	roboArmStates.stUInsertBackStart:		
		uInsertBack  := TRUE;
		resetActive  := TRUE;
		nextState(roboArmStates.stUInsertBackMove);				
		
// *** Unload Insert Back - Move
// Задава се програма на робота

	roboArmStates.stUInsertBackMove:		
		Stations.roboData := dataRequestRobot.roboPrg_PreUnload;		
		nextState(roboArmStates.stUInsertBackMoveCheck);		
		
// *** Unload Insert Back - Move Check
// Робота изпълни ли си хода ?

	roboArmStates.stUInsertBackMoveCheck:
		IF Stations.roboData = dataRequestRobot.done THEN				
		    nextState(roboArmStates.stUInsertBackSync);		
		END_IF		
		IF Stations.roboData = dataRequestRobot.error THEN
			nextState(roboArmStates.stErrRobot);
		END_IF
		timeOutError(robotMoveTime, roboArmStates.stErrRobotTimeOut);

// *** Unload Insert Back - Sync

	roboArmStates.stUInsertBackSync:	
		depWait(globalDeps.depULoadRobotOutOfRich);	     			
		nextState(roboArmStates.stUInsertBackDone);				
		
// *** Unload Insert Back - Done

	roboArmStates.stUInsertBackDone:
        uInsertBack	:= FALSE;
		nextState(roboArmStates.stUnloadStart);		
	
// *** Step Mode
		
	roboArmStates.stStepBlock:
		setDisplayState(roboArmDisplayStates.dStWaitForNextStep);
		
// *** Stop 
// Станията е деактивирана
	
	roboArmStates.stStop:
	
		initDone			  := FALSE; 			
		resetActive           := FALSE;                           
		nextMoveStart         := FALSE;                            
		moveToEmptyStart      := FALSE;                           
		emptyToUnloadStart    := FALSE;                           
		unloadPalletStart     := FALSE;                            
		loadPalletStart       := FALSE;                            
		emptyPosStart         := FALSE;                            
		loadStart             := FALSE;                            
		unloadStart           := FALSE;                            
		lInsertStart          := FALSE;                            
		lInsertLockStart      := FALSE;                 
		lInsertBack           := FALSE;             
		uInsertStart          := FALSE;                           
		uInsertLockStart      := FALSE;                          
		uInsertBack           := FALSE;         
		blockRunForLoad       := FALSE;
		
// *** ERRORS

// *** ERROR - Init Sensor
// При стартиране на програмата не трябва да има сензор в грипера на робота
		roboArmStates.stErrInitSensor:
			setDisplayState(roboArmDisplayStates.dStErrInitSensorInGrip);
			
// *** ERROR - Pallet On 24
// При стартиране на програмата не трябва да има тара на чакаща поз. HEX 24
		roboArmStates.stErrInitPalletOn24:
			setDisplayState(roboArmDisplayStates.dStErrInitPalletOnWaitPos24);			

// *** ERROR - Pallet On 27
// При стартиране на програмата не трябва да има тара на чакаща поз. HEX 27
		roboArmStates.stErrInitPalletOn27:
			setDisplayState(roboArmDisplayStates.dStErrInitPalletOnWaitPos27);		

// *** ERROR - Grip Not Open
// Гирипера на робота не е отворил навреме
		roboArmStates.stErrGripNotOpen:
			setDisplayState(roboArmDisplayStates.dStErrGripNotOpen);
	
// *** ERROR - Grip Not Close
// Гирипера на робота не е затворил навреме
		roboArmStates.stErrGripNotClose:
			setDisplayState(roboArmDisplayStates.dStErrGripNotClose);			
			
// *** ERROR - Rot Not turn 180
// Ротатора не е завъртял сензора на обратно (180 град.)
		roboArmStates.stErrRotNotTurn180:
			setDisplayState(roboArmDisplayStates.dStErrRotatorNotTurn180);			
			
// *** ERROR - Rot Not turn 0
// Ротатора не е завъртял сензора (0 град.)
		roboArmStates.stErrRotNotTurn0:
			setDisplayState(roboArmDisplayStates.dStErrRotatorNotTurn0);					
			
// *** ERROR - Slinde Not Down
// Слайдера който захваща тарата не в долна поз.
		roboArmStates.stErrSlliderNotDown:
			setDisplayState(roboArmDisplayStates.dStErrSlideNotDown);			
			
// *** ERROR - Slinde Not Up
// Слайдера който захваща тарата не в горна поз.
		roboArmStates.stErrSlideNotUp:
			setDisplayState(roboArmDisplayStates.dStErrSlideNotUp);	

// *** ERROR - Robot Error
// Има някаква грашка върната от робот контролера
		roboArmStates.stErrRobot:	
			setDisplayState(roboArmDisplayStates.dStErrRobotError);	
		
// *** ERROR - Robot Reset
// Времето за изпълнение на HOME програмата на работа е отнело трвърде мн.
		roboArmStates.stErrRobotReset:	
			setDisplayState(roboArmDisplayStates.dStErrRobotHomeMoveIsTooLong);			

// *** ERROR - Robot Time out
// Времето за изпълнение на движение на робота е отнело твърде мн.
		roboArmStates.stErrRobotTimeOut:	
			setDisplayState(roboArmDisplayStates.dStErrRobotMoveIsTooLong);	

// *** ERROR - Robot Recipe TimeOut
// Времето за зареждане на рецепта в робота е отнело твърде мн.
		roboArmStates.stErrRobotRecipeTimeOut:	
			setDisplayState(roboArmDisplayStates.dStErrRobotRecipeLoadIsTooLong);		
		
// *** ERROR - Robot Wait Pos Pallet Fail
// На мястото на чакащата поз. няма тара
		roboArmStates.stErrNoPalletWaitPos:	
			setDisplayState(roboArmDisplayStates.dStErrRobotWaitPosIsEmpty);	

// *** ERROR - Paallet On Wait Pos
// Робота трябва да занесе тара на чакаща поз, но там вече има
		roboArmStates.stErrPalletOnWaitPos:			
			setDisplayState(roboArmDisplayStates.dStErrRobotWaitPosIsNotEmpty);			
			
// *** ERROR - No Pallet Unload
// Робота не е могъл да вдигне или е изпуснал тара
		roboArmStates.stErrNoPalletUnload:	
			setDisplayState(roboArmDisplayStates.dStErrRobotNoPalletAtUnloadStacker);
			unloadPalletStart := FALSE;
			palletIn          := FALSE;	
			
// *** EMG State					
	roboArmStates.stEMG: 
		nextState(roboArmStates.stInit);

END_CASE

METHOD PRIVATE signalLamps
VAR_INPUT
	
	enable      : BOOL;                  
	lamp24      : BOOL;                  // Активиране на лампа за чакаща поз. за HEX 24
	sensor24    : BOOL;                  // Сигнал от сензора за поставена тара на поз. HEX 24
	lamp27      : BOOL;                  // Активиране на лампа за чакаща поз. за HEX 24	
	sensor27    : BOOL;                  // Сигнал от сензора за поставена тара на поз. HEX 27

END_VAR

VAR
	
	lamp24On    : BOOL;
	lamp27On    : BOOL;
	
END_VAR
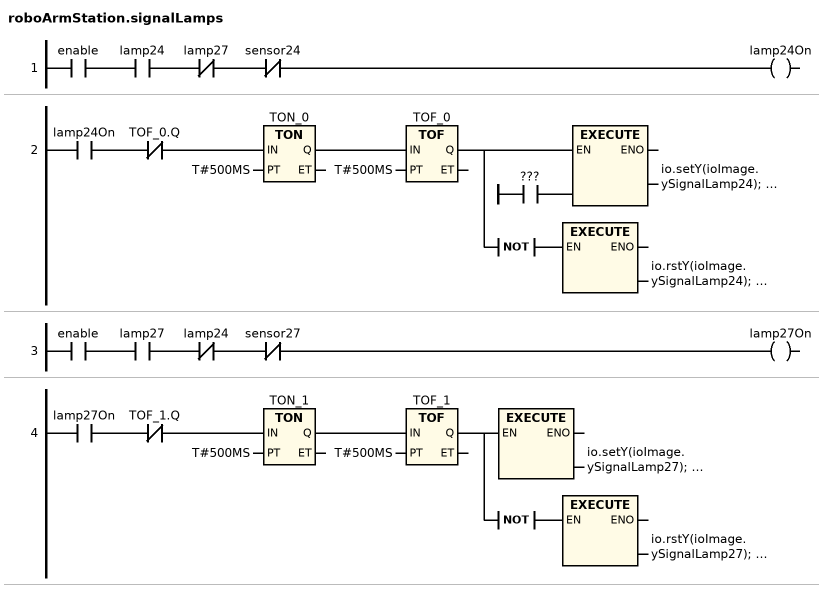
// NETWORK 1
lamp24On := enable AND lamp24 AND NOT lamp27 AND NOT sensor24;

// NETWORK 2
TON_0(IN := lamp24On AND NOT TOF_0.Q, PT := T#500MS); // TON
TOF_0(IN := TON_0.Q, PT := T#500MS); // TOF
IF TOF_0.Q THEN io.setY(ioImage.ySignalLamp24); END_IF
IF NOT TOF_0.Q THEN io.rstY(ioImage.ySignalLamp24); END_IF

// NETWORK 3
lamp27On := enable AND lamp27 AND NOT lamp24 AND NOT sensor27;

// NETWORK 4
TON_1(IN := lamp27On AND NOT TOF_1.Q, PT := T#500MS); // TON
TOF_1(IN := TON_1.Q, PT := T#500MS); // TOF
IF TOF_1.Q THEN io.setY(ioImage.ySignalLamp27); END_IF
IF NOT TOF_1.Q THEN io.rstY(ioImage.ySignalLamp27); END_IF
END_METHOD

END_FUNCTION_BLOCK

// ---- POUs/ROBOT.TcPOU
PROGRAM Robot
VAR
	fbRobot						: FB_Robot_Mitsubishi;
	nCurrentState				: DINT;
	nLastState					: DINT;				
	rtRobot_ProgramStarted		: TON;
	rtRobot_ProgramCompleted	: TON;
	fbTimerRobot				: TON;
	gbTimerTimeoutRobot			: TON;
END_VAR

Stations.gstRobotMitsubishi.sRobotAddress := '192.168.0.20';
Stations.gstRobotMitsubishi.nRobotPort := 10004;
Stations.gstRobotMitsubishi.bAutomaticMode := TRUE;
fbRobot(Robot := Stations.gstRobotMitsubishi,
	PacketManager := Stations.gstRobotMitsubishiPacketManager);
		
rtRobot_ProgramStarted(IN:=NOT Stations.gstRobotMitsubishi.bReady 
						AND NOT Stations.gstRobotMitsubishi.bProgramCompleted, PT:=T#30MS);
rtRobot_ProgramCompleted(IN:= Stations.gstRobotMitsubishi.bReady AND Stations.gstRobotMitsubishi.bProgramCompleted 
							AND Stations.gstRobotMitsubishi.nDependencyState = 0, PT:=T#30MS);

// If robot error
IF Stations.gstRobotMitsubishi.bError 
AND nCurrentState > E_RobotStates.STATE_INIT_CHECK_ROBOT_ERROR_DONE 
AND nCurrentState < E_RobotStates.STATE_ERROR THEN
	nLastState:=nCurrentState;
	nCurrentState:=E_RobotStates.STATE_ERROR;
END_IF
//Statuses
TagsRobot.robotError := Stations.gstRobotMitsubishi.bError;
TagsRobot.robotComOnline := Stations.gstRobotMitsubishi.bOnline;

// Robot Settings
Stations.gstRobotMitsubishi.nTargetProductID := TagsRobot.roboRecipeNum;
Stations.gstRobotMitsubishi.nTargetGripperID := 1;		//TBD Setting for GipperID
Stations.gstRobotMitsubishi.nTargetTrayOrientation := TagsRobot.rotPallet;
		
CASE nCurrentState OF
	E_RobotStates.STATE_WAITING_FOR_INIT:
		IF Stations.roboData = dataRequestRobot.roboInit THEN			
			nLastState := nCurrentState;
			nCurrentState := E_RobotStates.STATE_INIT_ROBOT_TOGGLE;
		END_IF
		
	E_RobotStates.STATE_INIT_ROBOT_TOGGLE:
		IF Stations.gstRobotMitsubishi.bAutomaticMode THEN
			Stations.gstRobotMitsubishi.bDoReset:=FALSE;
			Stations.gstRobotMitsubishi.bToggleConnect:=FALSE;
			Stations.gstRobotMitsubishi.bDoStart:=FALSE;
			fbTimerRobot(IN:=TRUE,PT:=T#1000MS);
			IF fbTimerRobot.Q THEN
				fbTimerRobot(IN:=FALSE);				
				nLastState := nCurrentState;
				nCurrentState :=E_RobotStates.STATE_INIT_ROBOT_ON;
			END_IF
		ELSE
			// Robot Auto  = true
		END_IF

	E_RobotStates.STATE_INIT_ROBOT_ON:
		IF Stations.gstRobotMitsubishi.bOnline THEN
			nLastState := nCurrentState;
			nCurrentState :=E_RobotStates.STATE_INIT_CHECK_ROBOT_ERROR;
		ELSE
			Stations.gstRobotMitsubishi.bToggleConnect:=TRUE;
			a_ToggleRobot();
		END_IF	

	E_RobotStates.STATE_INIT_CHECK_ROBOT_ERROR:
		IF Stations.gstRobotMitsubishi.bError OR Stations.gstRobotMitsubishi.nCurrentState = E_Robot_Mitsubishi_States.STATE_WAITING_RESET THEN
			Stations.gstRobotMitsubishi.bDoReset:=TRUE;
			nLastState := nCurrentState;
			nCurrentState :=E_RobotStates.STATE_INIT_CHECK_ROBOT_ERROR_DONE;
		ELSE
			nLastState := nCurrentState;
			nCurrentState :=E_RobotStates.STATE_INIT_CHECK_ROBOT_READY;
		END_IF	
	
	E_RobotStates.STATE_INIT_CHECK_ROBOT_ERROR_DONE:
		IF Stations.gstRobotMitsubishi.nCurrentState = E_Robot_Mitsubishi_States.STATE_OPERATIONAL THEN
			IF NOT Stations.gstRobotMitsubishi.bError THEN
				nLastState := nCurrentState;
				nCurrentState :=E_RobotStates.STATE_INIT_CHECK_ROBOT_READY;
			ELSE
				a_ToggleRobot();
			END_IF
		ELSIF Stations.gstRobotMitsubishi.nCurrentState = E_Robot_Mitsubishi_States.STATE_WAITING_RESET THEN
			nLastState := nCurrentState;
			nCurrentState :=E_RobotStates.STATE_INIT_CHECK_ROBOT_ERROR;
		END_IF
		
	E_RobotStates.STATE_INIT_CHECK_ROBOT_READY:
		IF NOT Stations.gstRobotMitsubishi.bReady OR NOT Stations.gstRobotMitsubishi.bExecuting THEN
			Stations.gstRobotMitsubishi.bDoStart:=TRUE;
			nLastState := nCurrentState;
			nCurrentState :=E_RobotStates.STATE_INIT_CHECK_ROBOT_READY_DONE;		
		ELSE
			nLastState := nCurrentState;
			nCurrentState :=E_RobotStates.STATE_INIT_CHECK_ROBOT_SERVOON;	
		END_IF
	
	E_RobotStates.STATE_INIT_CHECK_ROBOT_READY_DONE:
		IF Stations.gstRobotMitsubishi.bReady AND Stations.gstRobotMitsubishi.bExecuting THEN
			nLastState := nCurrentState;
			nCurrentState :=E_RobotStates.STATE_INIT_CHECK_ROBOT_SERVOON;
		ELSE
			a_ToggleRobot();					
		END_IF
				
	E_RobotStates.STATE_INIT_CHECK_ROBOT_SERVOON:		
		IF Stations.gstRobotMitsubishi.bPoweredOn AND Stations.gstRobotMitsubishi.bReady THEN
			nLastState := nCurrentState;
			nCurrentState :=E_RobotStates.STATE_INIT_DONE;
		ELSE 				
			Stations.gstRobotMitsubishi.bDoServoOn:=TRUE;
			nLastState := nCurrentState;
			nCurrentState :=E_RobotStates.STATE_INIT_CHECK_ROBOT_SERVOON_DONE;
		END_IF
		
	E_RobotStates.STATE_INIT_CHECK_ROBOT_SERVOON_DONE:
		IF Stations.gstRobotMitsubishi.bPoweredOn AND Stations.gstRobotMitsubishi.bReady THEN
			nLastState := nCurrentState;
			nCurrentState :=E_RobotStates.STATE_INIT_DONE;
		END_IF	
		
	E_RobotStates.STATE_INIT_DONE:
		Stations.roboData := dataRequestRobot.done;
		nLastState := nCurrentState;
		nCurrentState := E_RobotStates.STATE_WAITING_FOR_COMMAND;	
	
	E_RobotStates.STATE_WAITING_FOR_COMMAND:		
		IF Stations.roboData <> dataRequestRobot.done
		AND Stations.roboData <> dataRequestRobot.error 
		AND Stations.roboData <> dataRequestRobot.roboInit THEN
			Stations.gstRobotMitsubishi.nTargetProgram := Stations.roboData;
			IF Stations.roboData = dataRequestRobot.roboPrg_SensorLoad THEN
				Stations.gstRobotMitsubishi.nTargetTrayPosition := TagsRobot.loadPalletPos;
			ELSIF Stations.roboData = dataRequestRobot.roboPrg_SensorUnload THEN
				Stations.gstRobotMitsubishi.nTargetTrayPosition := TagsRobot.unLoadPalletPos;
			END_IF
			Stations.gstRobotMitsubishi.bDoStartProgram := TRUE;
			nLastState := nCurrentState;
			nCurrentState := E_RobotStates.STATE_WAITING_START_PRG;
		END_IF
		
	E_RobotStates.STATE_WAITING_START_PRG:
		IF rtRobot_ProgramStarted.Q THEN
			nLastState := nCurrentState;
			nCurrentState := E_RobotStates.STATE_PROGRAM_DONE;
		END_IF
		
	E_RobotStates.STATE_PROGRAM_DONE:
		IF rtRobot_ProgramCompleted.Q THEN
			Stations.roboData := dataRequestRobot.done;
			nLastState := nCurrentState;
			nCurrentState := E_RobotStates.STATE_WAITING_FOR_COMMAND;
		END_IF
		
	E_RobotStates.STATE_ERROR:
		Stations.roboData := dataRequestRobot.error;
		nLastState := nCurrentState;
		nCurrentState := E_RobotStates.STATE_WAITING_FOR_INIT;
		
END_CASE

ACTION a_ToggleRobot:
fbTimerRobot(IN:=TRUE,PT:=T#2000MS);
IF fbTimerRobot.Q THEN
	fbTimerRobot(IN:=FALSE);
	nLastState := nCurrentState;
	nCurrentState :=E_RobotStates.STATE_INIT_ROBOT_TOGGLE;
END_IF
END_ACTION

END_PROGRAM

// ---- POUs/Mitsubishi/FB_Robot_Mitsubishi.TcPOU
FUNCTION_BLOCK FB_Robot_Mitsubishi
VAR_INPUT
END_VAR
VAR_OUTPUT
END_VAR
VAR_IN_OUT
	Robot							: ST_Robot_Mitsubishi;											// Robot Mitsubishi station.	
	PacketManager					: ST_Robot_Misubishi_Packet_Manager;							// Robot Mitsubishi packet manager.
END_VAR
VAR
	nState							: E_Robot_Mitsubishi_States;	
	fbReceive						: FB_Robot_Mitsubishi_ReceivePacket;
	fbSend							: FB_Robot_Mitsubishi_SendPacket;	
	fbTimer							: TON;	
	fbStop							: R_TRIG;
	
	tResetTimeout					: TIME := T#5000MS;
	tPowerOnTimeout					: TIME := T#5000MS;
	tProgramStartTimeout			: TIME := T#2000MS;
	tProgramExecutionTimeout		: TIME := T#20000MS;
	tDependencyConfirmationTimeout	: TIME := T#20000MS;											// Should there be a timeout at all.
	tDependencyAcknoledgeTimeout	: TIME := T#5000MS;												//	|
	tChangeTargetStationTimeout		: TIME := T#5000MS;												//	|	Should be less than a seccond.
	tChangeTargetProgramTimeout		: TIME := T#5000MS;												//	|
	tChangeTargetSpeedTimeout		: TIME := T#5000MS;
	tChangeTargetCorrectionTimeout	: TIME := T#5000MS;
	tChangeStationTimeout			: TIME := T#2000MS;												//	|	Should be less than a seccond.
	tChangeProgramTimeout			: TIME := T#2000MS;												//	|
	tChangeSpeedTimeout				: TIME := T#2000MS;												//	|
	tChangeCorrectionTimeout		: TIME := T#2000MS;												//	|
	
	nDependencyReturnState			: E_Robot_Mitsubishi_States;									// The state to return to after confirming a dependency.
	
	bDisableTimeouts				: BOOL := TRUE;
	bAutoConfirm					: BOOL := FALSE;												// For testing while no connection is avalable.
	
	// TCP IP Connection.
	fbConnect 						: FB_ClientServerConnection;									// TCP IP Connection function block.
	sSrvNetID						: T_AmsNetID;													// TwinCAT TCP/IP server network address.
	eState							: E_SocketConnectionState := eSOCKET_DISCONNECTED;				// TCP/IP connection state.
	bDoConnect						: BOOL := FALSE;												//
	
	// CONTROL
	aOutputBuffer					: ARRAY[0..255] OF BYTE;										// The output command string sent to the robot.
	aInputBuffer					: ARRAY[0..255] OF BYTE;										// The output command string sent to the robot.
	fbSetOutputBuffer				: FB_SetOutputBuffer();											// Use to control the output buffer.
	fbClearOutputBuffer				: FB_ClearOutputBuffer();										// Use to cleanup the output buffer.	
	nLastRecPacketID				: DINT;
	sLastRecPacket					: STRING(255);	
	bBypassPacketSize				: BOOL := TRUE;	
	nRobotStateHolder				: DINT;	
	fbCompleted						: R_Trig;	
	wasFalse						: BOOL;
END_VAR

A_MonitorStop();
A_Connection();

fbSend( 
	ConnectionRef:= fbConnect, 
	nLastReceivedPacketID:= Robot.nLastReceivedPacketID,   
	bLastPacketConfirmed=> Robot.bLastPacketConfirmed);

//--------------------------------Check if robot is connected---------------------------------------
IF NOT Robot.bOnline THEN
	a_ResetAllRequests();
	fbSend(bDoSend:=FALSE);
	Robot.bReady := FALSE;
	Robot.bBusy := FALSE;
	Robot.bDisabled := TRUE;
	nState := E_Robot_Mitsubishi_States.STATE_OPERATIONAL;
ELSE	
	Robot.bDisabled := FALSE;
	CASE nState OF				
//----------------------------------OPERATIONAL----------------------------------------------------
		E_Robot_Mitsubishi_States.STATE_OPERATIONAL:							
			IF Robot.bError THEN
				a_ResetAllRequests();
				nState := E_Robot_Mitsubishi_States.STATE_ERROR_ROBOT;
			ELSE
				fbSend(bDoSend:=FALSE);
				IF Robot.bDoStart THEN
					nState := E_Robot_Mitsubishi_States.STATE_START_PROGRAM;								
				ELSIF Robot.bDoReset THEN
					nState := E_Robot_Mitsubishi_States.STATE_START_RESET;
				END_IF
				IF Robot.bReady THEN
					IF Robot.bDoServoOn THEN
						nState := E_Robot_Mitsubishi_States.STATE_START_POWER_ON;
					ELSIF Robot.bDoServoOff THEN
						nState := E_Robot_Mitsubishi_States.STATE_START_POWER_OFF;
					ELSIF Robot.bDoChangeTargetSpeed THEN
						nState := E_Robot_Mitsubishi_States.STATE_START_TARGET_SPEED_OVERRIDE_CHANGE;
					ELSIF Robot.bDoChangeTargetTrayPosition THEN
						nState := E_Robot_Mitsubishi_States.STATE_START_TARGET_TRAYPOS_CHANGE;					
					ELSIF Robot.bDoChangeTargetProgram THEN
						nState := E_Robot_Mitsubishi_States.STATE_START_TARGET_PROGRAM_CHANGE;
					ELSIF Robot.bDoStartProgram THEN
						nState := E_Robot_Mitsubishi_States.STATE_START_TARGET_PROGRAM;			
					ELSIF Robot.bDoOpenGripperA OR Robot.bDoCloseGripperA THEN
						nState := E_Robot_Mitsubishi_States.STATE_TOGGLE_GRIPERA;
					ELSIF Robot.bDoOpenGripperB OR Robot.bDoCloseGripperB THEN
						nState := E_Robot_Mitsubishi_States.STATE_TOGGLE_GRIPERB;
					END_IF
				ELSIF Robot.bExecuting THEN
					IF Robot.bDoStop THEN
						nState := E_Robot_Mitsubishi_States.STATE_START_STOP;								
					ELSIF Robot.bDoEnd <> Robot.bEnding THEN
						nState := E_Robot_Mitsubishi_States.STATE_SET_END;
					ELSIF Robot.bDoConfirmDependency AND Robot.nDependencyState <> 0 THEN
						nState := E_Robot_Mitsubishi_States.STATE_REQUEST_DEPENDENCY_CONFIRMATION;					
					END_IF
				END_IF
			END_IF
//------------------------------ START MAIN PROGRAM------------------------------------------------
		E_Robot_Mitsubishi_States.STATE_START_PROGRAM:
			A_SendStartProgram();		
			
		E_Robot_Mitsubishi_States.STATE_WAIT_PROGRAM_COMPLETED:			
			
//----------------------------------STOP-----------------------------------------------------------
		E_Robot_Mitsubishi_States.STATE_START_STOP:	
			A_SendStop();
			
		E_Robot_Mitsubishi_States.STATE_WAIT_STOP:
			IF (NOT Robot.bExecuting) THEN
				// STOPPED
				nState := E_Robot_Mitsubishi_States.STATE_STOPPED;
			END_IF
		E_Robot_Mitsubishi_States.STATE_STOPPED:
			IF (NOT Robot.bDoStop) THEN
				//A_SendStopReset();
				nState := E_Robot_Mitsubishi_States.STATE_OPERATIONAL;
			ELSE
				fbTimer(IN := TRUE, PT := tPowerOnTimeout);
				IF (fbTimer.Q AND (NOT bDisableTimeouts)) THEN
					A_ResetTimeoutTimer();
					nState := E_Robot_Mitsubishi_States.STATE_ERROR_STATE_MACHINE;
				ELSIF Robot.bError THEN
					A_ResetTimeoutTimer();
					nState := E_Robot_Mitsubishi_States.STATE_ERROR_ROBOT;
				END_IF
			END_IF
//----------------------------------END------------------------------------------------------------
		E_Robot_Mitsubishi_States.STATE_SET_END:
			A_SendSetEnd();	
		
		E_Robot_Mitsubishi_States.STATE_WAIT_SET_END:
			IF Robot.bEnding = Robot.bDoEnd THEN
				A_ResetTimeoutTimer();
				nState := E_Robot_Mitsubishi_States.STATE_OPERATIONAL;
			ELSE
				fbTimer(IN := TRUE, PT := tPowerOnTimeout);
				IF (fbTimer.Q AND (NOT bDisableTimeouts)) THEN
					A_ResetTimeoutTimer();
					nState := E_Robot_Mitsubishi_States.STATE_ERROR_STATE_MACHINE;
				ELSIF Robot.bError THEN
					A_ResetTimeoutTimer();
					nState := E_Robot_Mitsubishi_States.STATE_ERROR_ROBOT;
				END_IF
			END_IF
// ------------------------------ RESET -----------------------------------------------------------
		E_Robot_Mitsubishi_States.STATE_WAITING_RESET:
			IF Robot.bDoReset THEN
				nState := E_Robot_Mitsubishi_States.STATE_START_RESET;
			END_IF
			
		E_Robot_Mitsubishi_States.STATE_START_RESET:
			A_SendReset();
		
		E_Robot_Mitsubishi_States.STATE_WAITING_RESET_COMPLETED:
			fbTimer(IN := TRUE, PT := tResetTimeout);
			IF (NOT Robot.bError) THEN
				A_ResetTimeoutTimer();
				nState := E_Robot_Mitsubishi_States.STATE_OPERATIONAL;
			ELSIF (fbTimer.Q ) THEN
				A_ResetTimeoutTimer();
				nState := E_Robot_Mitsubishi_States.STATE_OPERATIONAL;
			END_IF
// ------------------------------ Power ON --------------------------------------------------------
		E_Robot_Mitsubishi_States.STATE_START_POWER_ON:
			A_SendPowerOn();
			
		E_Robot_Mitsubishi_States.STATE_WAIT_POWERED_ON:
			IF Robot.bPoweredOn THEN
				A_ResetTimeoutTimer();
				nState := E_Robot_Mitsubishi_States.STATE_OPERATIONAL;
			ELSE
				fbTimer(IN := TRUE, PT := tPowerOnTimeout);
				IF (fbTimer.Q AND (NOT bDisableTimeouts)) THEN
					A_ResetTimeoutTimer();
					nState := E_Robot_Mitsubishi_States.STATE_ERROR_STATE_MACHINE;
				ELSIF Robot.bError THEN
					A_ResetTimeoutTimer();
					nState := E_Robot_Mitsubishi_States.STATE_ERROR_ROBOT;
				END_IF
			END_IF
// ------------------------------ Power OFF -------------------------------------------------------
		E_Robot_Mitsubishi_States.STATE_START_POWER_OFF:
			A_SendPowerOff();
			
		E_Robot_Mitsubishi_States.STATE_WAIT_POWERED_OFF:
			IF (NOT Robot.bPoweredOn) THEN
				A_ResetTimeoutTimer();
				nState := E_Robot_Mitsubishi_States.STATE_OPERATIONAL;
			ELSE
				fbTimer(IN := TRUE, PT := tPowerOnTimeout);
				IF (fbTimer.Q AND (NOT bDisableTimeouts)) THEN
					A_ResetTimeoutTimer();
					nState := E_Robot_Mitsubishi_States.STATE_ERROR_STATE_MACHINE;
				ELSIF Robot.bError THEN
					A_ResetTimeoutTimer();
					nState := E_Robot_Mitsubishi_States.STATE_ERROR_ROBOT;
				END_IF
			END_IF
// ------------------------------ Dependency ------------------------------------------------------
		E_Robot_Mitsubishi_States.STATE_REQUEST_DEPENDENCY_CONFIRMATION:
			A_ResetTimeoutTimer();
			A_SendDependencyConfirmation();
			
		E_Robot_Mitsubishi_States.STATE_WAIT_DEPENDENCY_CONFIRMATION:
			// Could use the wait program active since it's the same.									// TODO: Probably better to return to the actual program execution monitoring.
			IF Robot.nDependencyState <> PacketManager.StateConfirmationPacket.StateID OR
				Robot.nDependencyState = 0 THEN
				A_ResetTimeoutTimer();
				nState := E_Robot_Mitsubishi_States.STATE_OPERATIONAL;												// Return to program execution.
			ELSE
				fbTimer(IN := TRUE, PT := tDependencyAcknoledgeTimeout);
				IF (fbTimer.Q AND (NOT bDisableTimeouts)) THEN
					A_ResetTimeoutTimer();
					nState := E_Robot_Mitsubishi_States.STATE_ERROR_STATE_MACHINE;
				ELSIF Robot.bError THEN
					A_ResetTimeoutTimer();
					nState := E_Robot_Mitsubishi_States.STATE_ERROR_ROBOT;
				END_IF
			END_IF
						
// ------------------------------ Settings --------------------------------------------------------
		E_Robot_Mitsubishi_States.STATE_START_TARGET_SPEED_OVERRIDE_CHANGE:
			a_SendChangeTargetSpeed();			

		E_Robot_Mitsubishi_States.STATE_START_TARGET_TRAYPOS_CHANGE:
			a_SendChangeCurrentTrayPosition();
		
		E_Robot_Mitsubishi_States.STATE_START_TARGET_PROGRAM_CHANGE:
			a_SendChangeCurrentProgram();
			
		E_Robot_Mitsubishi_States.STATE_START_TARGET_PROGRAM:
			a_SendChangeStartProgram();
			
		E_Robot_Mitsubishi_States.STATE_WAIT_PROGRAM_STARTED:
			IF NOT Robot.bReady THEN
				Robot.bDoStartProgram := FALSE;
				nState := E_Robot_Mitsubishi_States.STATE_OPERATIONAL;
			END_IF
			
		E_Robot_Mitsubishi_States.STATE_TOGGLE_GRIPERA:
			A_SendToggleGripperA();
			
		E_Robot_Mitsubishi_States.STATE_TOGGLE_GRIPERB:
			A_SendToggleGripperB();
// ------------------------------ ERROR -----------------------------------------------------------
		E_Robot_Mitsubishi_States.STATE_ERROR_ROBOT:
			// Handle any error???
			a_ResetAllRequests();
			nState := E_Robot_Mitsubishi_States.STATE_WAITING_RESET;
			
		E_Robot_Mitsubishi_States.STATE_ERROR_STATE_MACHINE:
			;
		
	END_CASE
	
END_IF
IF (nState <> Robot.nCurrentState) THEN
	Robot.nLastState := Robot.nCurrentState;
	Robot.nCurrentState := nState;
	IF ((nState = E_Robot_Mitsubishi_States.STATE_ERROR_ROBOT) OR
		(nState = E_Robot_Mitsubishi_States.STATE_ERROR_STATE_MACHINE)) THEN
		Robot.nLastErrorState := Robot.nLastState;
	END_IF
END_IF
A_ParseInput();

ACTION A_Connection:
fbConnect( 	sSrvNetID 		:= sSrvNetID,
		nMode			:= SEL( TRUE, 0, CONNECT_MODE_ENABLEDBG),
		sRemoteHost 	:= Robot.sRobotAddress,		
		nRemotePort 	:= Robot.nRobotPort,
		bEnable			:= Robot.bToggleConnect,
		eState			=> eState );
		
Robot.bOnline := eState = eSOCKET_CONNECTED;
END_ACTION

ACTION A_MonitorStop:
fbStop(CLK := Robot.bDoStop);

IF fbStop.Q AND Robot.bExecuting THEN
	nState := E_Robot_Mitsubishi_States.STATE_START_STOP;
END_IF
END_ACTION

ACTION A_ParseInput:
// SWITCH ReceivedPacket.0 AS ID :
fbReceive(LastReceivedPacket => sLastRecPacket,
	LastReceivedPacketID => nLastRecPacketID,
	ConnectionRef := fbConnect);
IF LEN(sLastRecPacket) > 0 THEN
	CASE nLastRecPacketID OF
		1000:
			// Robot status packet.
			IF (((SIZEOF(PacketManager.StatusPacket) + 2) = LEN(sLastRecPacket)) OR bBypassPacketSize) THEN
				A_ParseStatusPacket();			
			ELSE
				// ERROR
				// SIZEOF StatusPacket is wrong.
			END_IF
			
		1100:
			// Robot correction packet.
			
		1101:
			// Robot packet confirmation packet.
			IF (((SIZEOF(PacketManager.PacketConfirmationPacket) + 2) = LEN(sLastRecPacket)) OR bBypassPacketSize) THEN
				A_ParsePacketConfirmationPacket();
			ELSE
				// ERROR
				// SIZEOF StatusPacket is wrong.
			END_IF		
		ELSE
			sLastRecPacket := '';																			// Always cleanup.
	END_CASE
	MEMSET(ADR(sLastRecPacket),
		0,
		SIZEOF(sLastRecPacket));
END_IF
END_ACTION

ACTION A_ParsePacketConfirmationPacket:
FB_HEXSTR_TO_DINT(in := LEFT(RIGHT(sLastRecPacket, LEN(sLastRecPacket) - 8), 8),
	out => PacketManager.PacketConfirmationPacket.LastReceivedPacketID);

Robot.nLastReceivedPacketID := PacketManager.PacketConfirmationPacket.LastReceivedPacketID;
END_ACTION

ACTION A_ParseStatusPacket:
sLastRecPacket := RIGHT(sLastRecPacket, LEN(sLastRecPacket) - 8);
FB_HEXSTR_TO_DINT(in := LEFT(sLastRecPacket, 8),
	out => nRobotStateHolder);

PacketManager.StatusPacket.Ready := nRobotStateHolder.15;
PacketManager.StatusPacket.Busy := nRobotStateHolder.14;
PacketManager.StatusPacket.Error := nRobotStateHolder.13;
PacketManager.StatusPacket.PoweredOn := nRobotStateHolder.12;
PacketManager.StatusPacket.AutomaticMode := nRobotStateHolder.11;
PacketManager.StatusPacket.Executing := nRobotStateHolder.10;
PacketManager.StatusPacket.Ending := nRobotStateHolder.9;
PacketManager.StatusPacket.ProgramCompleted := nRobotStateHolder.8;
PacketManager.StatusPacket.GripperA_Present := nRobotStateHolder.7;
PacketManager.StatusPacket.GripperB_Present := nRobotStateHolder.6;
PacketManager.StatusPacket.GripperA_Open := nRobotStateHolder.5;
PacketManager.StatusPacket.GripperB_Open := nRobotStateHolder.4;
	
Robot.bReady := (PacketManager.StatusPacket.Ready AND 
(nState = E_Robot_Mitsubishi_States.STATE_OPERATIONAL));
Robot.bBusy := PacketManager.StatusPacket.Busy;
Robot.bError := PacketManager.StatusPacket.Error;
Robot.bPoweredOn := PacketManager.StatusPacket.PoweredOn;
//Robot.bAutomaticMode := PacketManager.StatusPacket.AutomaticMode;
Robot.bExecuting := PacketManager.StatusPacket.Executing;
Robot.bEnding := PacketManager.StatusPacket.Ending;
Robot.bProgramCompleted := Robot.nCurrentProgram = Robot.nTargetProgram AND PacketManager.StatusPacket.ProgramCompleted;
Robot.bGripperAPresent	:= NOT PacketManager.StatusPacket.GripperA_Present;
Robot.bGripperBPresent	:= NOT PacketManager.StatusPacket.GripperB_Present;

sLastRecPacket := RIGHT(sLastRecPacket, LEN(sLastRecPacket) - 8);
FB_HEXSTR_TO_DINT(in := LEFT(sLastRecPacket, 8),
	out => PacketManager.StatusPacket.CurrentState);
	
sLastRecPacket := RIGHT(sLastRecPacket, LEN(sLastRecPacket) - 8);
FB_HEXSTR_TO_DINT(in := LEFT(sLastRecPacket, 8),
	out => PacketManager.StatusPacket.CurrentProgram);
	
sLastRecPacket := RIGHT(sLastRecPacket, LEN(sLastRecPacket) - 8);
FB_HEXSTR_TO_DINT(in := LEFT(sLastRecPacket, 8),
	out => PacketManager.StatusPacket.CurrentTrayPosition);
	
sLastRecPacket := RIGHT(sLastRecPacket, LEN(sLastRecPacket) - 8);
FB_HEXSTR_TO_DINT(in := LEFT(sLastRecPacket, 8),
	out => PacketManager.StatusPacket.CurrentSpeed);
	
sLastRecPacket := RIGHT(sLastRecPacket, LEN(sLastRecPacket) - 8);
//Product ID
FB_HEXSTR_TO_DINT(in := LEFT(sLastRecPacket, 8),
	out => PacketManager.StatusPacket.CurrentProductID);
	
sLastRecPacket := RIGHT(sLastRecPacket, LEN(sLastRecPacket) - 8);
FB_HEXSTR_TO_DINT(in := LEFT(sLastRecPacket, 8),
	out => PacketManager.StatusPacket.CurrentGripperID);
	
sLastRecPacket := RIGHT(sLastRecPacket, LEN(sLastRecPacket) - 8);
FB_HEXSTR_TO_DINT(in := LEFT(sLastRecPacket, 8),
	out => PacketManager.StatusPacket.CurrentTrayOrient);
	
sLastRecPacket := RIGHT(sLastRecPacket, LEN(sLastRecPacket) - 8);
FB_HEXSTR_TO_DINT(in := LEFT(sLastRecPacket, 8),
	out => PacketManager.StatusPacket.CurrentTargetProgram);
	
sLastRecPacket := RIGHT(sLastRecPacket, LEN(sLastRecPacket) - 8);
FB_HEXSTR_TO_DINT(in := LEFT(sLastRecPacket, 8),
	out => PacketManager.StatusPacket.CurrentTargetTrayPosition);
	
sLastRecPacket := RIGHT(sLastRecPacket, LEN(sLastRecPacket) - 8);
FB_HEXSTR_TO_DINT(in := LEFT(sLastRecPacket, 8),
	out => PacketManager.StatusPacket.CurrentTargetSpeed);
// ----
sLastRecPacket := RIGHT(sLastRecPacket, LEN(sLastRecPacket) - 8);
FB_HEXSTR_TO_DINT(in := LEFT(sLastRecPacket, 8),
	out => PacketManager.StatusPacket.CurrentTargetProductID);
	
sLastRecPacket := RIGHT(sLastRecPacket, LEN(sLastRecPacket) - 8);
FB_HEXSTR_TO_DINT(in := LEFT(sLastRecPacket, 8),
	out => PacketManager.StatusPacket.CurrentTargetGripperID);
	
sLastRecPacket := RIGHT(sLastRecPacket, LEN(sLastRecPacket) - 8);
FB_HEXSTR_TO_DINT(in := LEFT(sLastRecPacket, 8),
	out => PacketManager.StatusPacket.CurrentTargetTrayOrient);

Robot.nDependencyState := PacketManager.StatusPacket.CurrentState;
Robot.nCurrentProgram := PacketManager.StatusPacket.CurrentProgram;
Robot.nCurrentTrayPosition := PacketManager.StatusPacket.CurrentTrayPosition;
Robot.nCurrentSpeed := PacketManager.StatusPacket.CurrentSpeed;
Robot.nCurrentProductID := PacketManager.StatusPacket.CurrentProductID;
Robot.nCurrentGripperID := PacketManager.StatusPacket.CurrentGripperID;
Robot.nCurrentTrayOrient := PacketManager.StatusPacket.CurrentTrayOrient;

Robot.nCurrentTargetProgram := PacketManager.StatusPacket.CurrentTargetProgram;
Robot.nCurrentTargetTrayPosition := PacketManager.StatusPacket.CurrentTargetTrayPosition;
Robot.nCurrentTargetSpeed := PacketManager.StatusPacket.CurrentTargetSpeed;
Robot.nCurrentTargetProductID := PacketManager.StatusPacket.CurrentTargetProductID;
Robot.nCurrentTargetGripperID := PacketManager.StatusPacket.CurrentTargetGripperID;
Robot.nCurrentTargetTrayOrient := PacketManager.StatusPacket.CurrentTargetTrayOrient;
END_ACTION

ACTION A_ResetAllRequests:
// Robot Requests
Robot.bDoOpenGripperB := FALSE;
Robot.bDoCloseGripperB := FALSE;
Robot.bDoOpenGripperB := FALSE;
Robot.bDoCloseGripperB := FALSE;
Robot.bDoServoOn := FALSE;
Robot.bDoServoOff := FALSE;
Robot.bDoStart := FALSE;
Robot.bDoStop := FALSE;
Robot.bDoEnd := FALSE;
Robot.bDoReset:=FALSE;
Robot.bDoStepFwd := FALSE;
Robot.bDoStepBwd := FALSE;
Robot.bDoChangeTargetProgram := FALSE;
Robot.bDoChangeTargetSpeed := FALSE;
Robot.bDoChangeTargetTrayPosition := FALSE;
Robot.bDoChangeTargetCorrection := FALSE;
Robot.bDoOpenGripperA:=FALSE;
Robot.bDoCloseGripperA:=FALSE;
Robot.bDoOpenGripperB:=FALSE;
Robot.bDoCloseGripperB:=FALSE;
Robot.bDoConfirmDependency := FALSE;
Robot.bDoStartProgram :=FALSE;

//Control Package bits -! Very important!
PacketManager.ControlPacket.Reset := FALSE;
PacketManager.ControlPacket.Start := FALSE;
PacketManager.ControlPacket.Stop := FALSE;
PacketManager.ControlPacket.ServoOn := FALSE;
PacketManager.ControlPacket.ServoOff := FALSE;
PacketManager.ControlPacket.OpenGripperA := FALSE;
PacketManager.ControlPacket.CloseGripperA := FALSE;
PacketManager.ControlPacket.OpenGripperB := FALSE;
PacketManager.ControlPacket.CloseGripperB := FALSE;
PacketManager.ControlPacket.End := FALSE;
PacketManager.SettingsPacket.StartProgram := FALSE;
END_ACTION

ACTION A_ResetTimeoutTimer:
fbTimer(IN := FALSE);
END_ACTION

ACTION a_SendChangeCurrentProgram:
PacketManager.SettingsPacket.TargetProgram := Robot.nTargetProgram;

fbSend(PacketAddress := ADR(PacketManager.SettingsPacket),
	SizeOfPacket := SIZEOF(PacketManager.SettingsPacket),
	bDoSend := TRUE);
	
// ALWAYS CLEANUP IF NECCESSARY
IF fbSend.bLastPacketConfirmed THEN
	fbSend(bDoSend:=FALSE);
	a_ResetAllRequests();
	nState := E_Robot_Mitsubishi_States.STATE_OPERATIONAL;
END_IF
END_ACTION

ACTION a_SendChangeCurrentTrayPosition:
PacketManager.SettingsPacket.TargetTrayPosition := Robot.nTargetTrayPosition;

fbSend(PacketAddress := ADR(PacketManager.SettingsPacket),
	SizeOfPacket := SIZEOF(PacketManager.SettingsPacket),
	bDoSend := TRUE);
	
// ALWAYS CLEANUP IF NECCESSARY
IF fbSend.bLastPacketConfirmed THEN
	fbSend(bDoSend:=FALSE);
	a_ResetAllRequests();
	nState := E_Robot_Mitsubishi_States.STATE_OPERATIONAL;
END_IF
END_ACTION

ACTION a_SendChangeStartProgram:
PacketManager.SettingsPacket.StartProgram := TRUE;
PacketManager.SettingsPacket.TargetProgram := Robot.nTargetProgram;
PacketManager.SettingsPacket.TargetTrayPosition := Robot.nTargetTrayPosition;
PacketManager.SettingsPacket.TargetSpeed := Robot.nTargetSpeed;
PacketManager.SettingsPacket.TargetProductID := Robot.nTargetProductID;
PacketManager.SettingsPacket.TargetGripperID := Robot.nTargetGripperID;
PacketManager.SettingsPacket.TargetTrayOrientation := Robot.nTargetTrayOrientation;


fbSend(PacketAddress := ADR(PacketManager.SettingsPacket),
	SizeOfPacket := SIZEOF(PacketManager.SettingsPacket),
	bDoSend := TRUE);
	
fbTimer(IN:=TRUE,PT:=T#1000MS);
// ALWAYS CLEANUP IF NECCESSARY
IF fbSend.bLastPacketConfirmed THEN
	fbSend(bDoSend:=FALSE);	
	fbTimer(IN := FALSE);
	a_ResetAllRequests();
	nState := E_Robot_Mitsubishi_States.STATE_WAIT_PROGRAM_STARTED;	
ELSIF fbTimer.Q AND NOT fbSend.bLastPacketConfirmed THEN
	fbTimer(IN := FALSE);
	a_ResetAllRequests();
	nState := E_Robot_Mitsubishi_States.STATE_OPERATIONAL;
END_IF
END_ACTION

ACTION a_SendChangeTargetSpeed:
PacketManager.SettingsPacket.TargetSpeed := Robot.nTargetSpeed;

fbSend(PacketAddress := ADR(PacketManager.SettingsPacket),
	SizeOfPacket := SIZEOF(PacketManager.SettingsPacket),
	bDoSend := TRUE);
	
// ALWAYS CLEANUP IF NECCESSARY
IF fbSend.bLastPacketConfirmed THEN
	fbSend(bDoSend:=FALSE);
	a_ResetAllRequests();
	nState := E_Robot_Mitsubishi_States.STATE_OPERATIONAL;
END_IF
END_ACTION

ACTION A_SendDependencyConfirmation:
PacketManager.StateConfirmationPacket.StateID := Robot.nDependencyState;					// TODO: Should be outer set to be properly used.

fbSend(PacketAddress := ADR(PacketManager.StateConfirmationPacket),
	SizeOfPacket := SIZEOF(PacketManager.StateConfirmationPacket),
	bDoSend := TRUE);
	
// ALWAYS CLEANUP IF NECCESSARY
	
IF fbSend.bLastPacketConfirmed 
OR (Robot.nDependencyState = 0) THEN
	fbSend(bDoSend:=FALSE);
	IF NOT Robot.bDoConfirmDependency THEN
		Global.gnLostDPPackets := Global.gnLostDPPackets + 1;
	END_IF
	a_ResetAllRequests();
	nState := E_Robot_Mitsubishi_States.STATE_WAIT_DEPENDENCY_CONFIRMATION;		// Go to wait confirmation acknowledge.
	A_ResetTimeoutTimer();
END_IF
END_ACTION

ACTION A_SendPowerOff:
PacketManager.ControlPacket.ServoOff := TRUE;

fbSend(PacketAddress := ADR(PacketManager.ControlPacket),
	SizeOfPacket := SIZEOF(PacketManager.ControlPacket),
	bDoSend := TRUE);
	
// ALWAYS CLEANUP IF NECCESSARY
IF fbSend.bLastPacketConfirmed THEN
	fbSend(bDoSend:=FALSE);
	a_ResetAllRequests();
	nState := E_Robot_Mitsubishi_States.STATE_WAIT_POWERED_OFF;
	fbTimer(IN := FALSE);
END_IF
END_ACTION

ACTION A_SendPowerOn:
PacketManager.ControlPacket.ServoOn := TRUE;
fbTimer(IN := TRUE, PT := tPowerOnTimeout);

fbSend(PacketAddress := ADR(PacketManager.ControlPacket),
	SizeOfPacket := SIZEOF(PacketManager.ControlPacket),
	bDoSend := TRUE);
	
// ALWAYS CLEANUP IF NECCESSARY
IF fbSend.bLastPacketConfirmed THEN
	fbSend(bDoSend:=FALSE);
	a_ResetAllRequests();
	nState := E_Robot_Mitsubishi_States.STATE_WAIT_POWERED_ON;
	fbTimer(IN := FALSE);
ELSIF fbTimer.Q THEN
	fbSend(bDoSend:=FALSE);
	a_ResetAllRequests();
	fbTimer(IN := FALSE);
	nState := E_Robot_Mitsubishi_States.STATE_OPERATIONAL;
END_IF
END_ACTION

ACTION A_SendReset:
PacketManager.ControlPacket.Reset := TRUE;

fbSend(PacketAddress := ADR(PacketManager.ControlPacket),
	SizeOfPacket := SIZEOF(PacketManager.ControlPacket),
	bDoSend := TRUE);
	
// ALWAYS CLEANUP IF NECCESSARY
IF fbSend.bLastPacketConfirmed THEN
	fbSend(bDoSend:=FALSE);
	fbTimer(IN := FALSE);
	a_ResetAllRequests();
	nState := E_Robot_Mitsubishi_States.STATE_WAITING_RESET_COMPLETED;	
END_IF
END_ACTION

ACTION A_SendSetEnd:
PacketManager.ControlPacket.End := TRUE;

fbSend(PacketAddress := ADR(PacketManager.ControlPacket),
	SizeOfPacket := SIZEOF(PacketManager.ControlPacket),
	bDoSend := TRUE);
	
// ALWAYS CLEANUP IF NECCESSARY
IF fbSend.bLastPacketConfirmed THEN
	fbSend(bDoSend:=FALSE);
	a_ResetAllRequests();
	fbTimer(IN := FALSE);
	nState := E_Robot_Mitsubishi_States.STATE_WAIT_SET_END;	
END_IF
END_ACTION

ACTION a_SendStartProgram:
PacketManager.ControlPacket.Start := TRUE;

fbSend(PacketAddress := ADR(PacketManager.ControlPacket),
	SizeOfPacket := SIZEOF(PacketManager.ControlPacket),
	bDoSend := TRUE);
	
// ALWAYS CLEANUP IF NECCESSARY
IF fbSend.bLastPacketConfirmed THEN
	fbSend(bDoSend:=FALSE);
	a_ResetAllRequests();
	nState := E_Robot_Mitsubishi_States.STATE_OPERATIONAL;
	fbTimer(IN := FALSE);
END_IF
END_ACTION

ACTION A_SendStop:
PacketManager.ControlPacket.Stop := TRUE;

fbSend(PacketAddress := ADR(PacketManager.ControlPacket),
	SizeOfPacket := SIZEOF(PacketManager.ControlPacket),
	bDoSend := TRUE);
	
// ALWAYS CLEANUP IF NECCESSARY
IF fbSend.bLastPacketConfirmed THEN
	fbSend(bDoSend:=FALSE);
	a_ResetAllRequests();
	nState := E_Robot_Mitsubishi_States.STATE_WAIT_STOP;
	fbTimer(IN := FALSE);
END_IF
END_ACTION

ACTION A_SendToggleGripperA:
PacketManager.ControlPacket.OpenGripperA := Robot.bDoOpenGripperA;
PacketManager.ControlPacket.CloseGripperA := Robot.bDoCloseGripperA;


fbSend(PacketAddress := ADR(PacketManager.ControlPacket),
	SizeOfPacket := SIZEOF(PacketManager.ControlPacket),
	bDoSend := TRUE);

// ALWAYS CLEANUP IF NECCESSARY
IF fbSend.bLastPacketConfirmed THEN
	fbSend(bDoSend:=FALSE);
	a_ResetAllRequests();
	nState := E_Robot_Mitsubishi_States.STATE_OPERATIONAL;
END_IF
END_ACTION

ACTION A_SendToggleGripperB:
PacketManager.ControlPacket.OpenGripperB := Robot.bDoOpenGripperB;
PacketManager.ControlPacket.CloseGripperB := Robot.bDoCloseGripperB;

fbSend(PacketAddress := ADR(PacketManager.ControlPacket),
	SizeOfPacket := SIZEOF(PacketManager.ControlPacket),
	bDoSend := TRUE);

// ALWAYS CLEANUP IF NECCESSARY
IF fbSend.bLastPacketConfirmed THEN
	fbSend(bDoSend:=FALSE);
	a_ResetAllRequests();
	nState := E_Robot_Mitsubishi_States.STATE_OPERATIONAL;
END_IF
END_ACTION

END_FUNCTION_BLOCK

// ---- POUs/Mitsubishi/FB_Robot_Mitsubishi_ReceivePacket.TcPOU
FUNCTION_BLOCK FB_Robot_Mitsubishi_ReceivePacket
VAR_INPUT
END_VAR
VAR_OUTPUT
	LastReceivedPacket				: STRING(255);
	LastReceivedPacketID			: DINT;
END_VAR
VAR_IN_OUT
	ConnectionRef					: FB_ClientServerConnection;											//
END_VAR
VAR
	fbReceive						: FB_SocketReceive;														// Receive data trough TCP IP.
	aInputBuffer					: ARRAY[0..255] OF BYTE;												// 
	bBusy							: BOOL;
END_VAR

IF ConnectionRef.eState = eSOCKET_CONNECTED AND (NOT ConnectionRef.bBusy) THEN
	IF NOT bBusy THEN
		fbReceive( bExecute := FALSE);	
		fbReceive( 	sSrvNetId	:= ConnectionRef.sSrvNetID,
					hSocket		:= ConnectionRef.hSocket,
					cbLen		:= SIZEOF(aInputBuffer),
					pDest		:= ADR(aInputBuffer),
					tTimeout	:= T#100MS,
					bExecute	:= TRUE);
		bBusy := TRUE;
	ELSE
		fbReceive( bExecute := FALSE);
		IF (NOT fbReceive.bBusy) THEN
			bBusy := FALSE;
			IF fbReceive.nRecBytes > 10 THEN															// 8 Bytes for packet ID and 2 bytes for <LF><CR>
				LastReceivedPacketID := 0;
				LastReceivedPacket := '';
				MEMCPY(ADR(LastReceivedPacket),														// Copy the packet header data.
					ADR(aInputBuffer),																// Could trim the <LF><CR> flags.
					fbReceive.nRecBytes);
				FB_HEXSTR_TO_DINT(in := LEFT(LastReceivedPacket, 8),
					out => LastReceivedPacketID);
				MEMSET(ADR(aInputBuffer),
					0,
					SIZEOF(aInputBuffer));
			ELSE
				MEMSET(ADR(aInputBuffer),
					0,
					SIZEOF(aInputBuffer));
			END_IF
		END_IF
	END_IF
ELSE
	fbReceive( bExecute := FALSE );
END_IF

END_FUNCTION_BLOCK

// ---- POUs/Mitsubishi/Func/FB_HEXSTR_TO_DINT.TcPOU
FUNCTION FB_HEXSTR_TO_DINT																			// Converts a STRING hex array to DINT.
VAR_INPUT
	in						: STRING;																// The input string.
END_VAR
VAR_OUTPUT
	out						: DINT;																	// The output value.
	bError					: BOOL;																	// Had any error occured.
END_VAR
VAR
	sSum					: STRING;
	pVal					: PVOID;
END_VAR

// Converts a STRING hex array to DINT.
IF LEN(in) = 8 THEN
	sSum := CONCAT('16#', in);
	pVal := STRING_TO_PVOID(sSum);
	MEMCPY(ADR(out),
		ADR(pVal),
		4);
ELSE
	out := 0;
	bError := TRUE;
END_IF

END_FUNCTION

// ---- POUs/Mitsubishi/FB_Robot_Mitsubishi_SendPacket.TcPOU
FUNCTION_BLOCK FB_Robot_Mitsubishi_SendPacket
VAR_INPUT
	PacketAddress					: PVOID;
	SizeOfPacket					: UDINT;
	bDoSend							: BOOL;
	ConnectionRef					: FB_ClientServerConnection;
	nLastReceivedPacketID			: DINT;
END_VAR
VAR_OUTPUT
	bLastPacketConfirmed			: BOOL;
END_VAR
VAR_IN_OUT

END_VAR
VAR
	fbSend							: FB_SocketSend;// Send data trought TCP IP.
	fbTimerSend						: TON;								
	eState							: E_Communication_Send_States;
	nPacketLenght					: UDINT;
	
	sOutputString					: STRING(255);
	nCounter						: UDINT;
	nLastSentPacketID				: DINT;
END_VAR

// This should all be a state machine.
fbSend(sSrvNetID 	:= ConnectionRef.sSrvNetID,
			hSocket		:= ConnectionRef.hSocket);
			
IF NOT (bDoSend) THEN
	bLastPacketConfirmed := FALSE;													// Reset the confirmation flag.
	nLastReceivedPacketID := 0;
	sOutputString := '';
	fbSend(bExecute	:= FALSE);	
	eState := E_Communication_Send_States.E_COM_SEND_PREPARE;
ELSE
	CASE eState OF
		E_Communication_Send_States.E_COM_SEND_PREPARE:			
			FOR nCounter := 0 TO SizeOfPacket - 4 BY 4 DO
				sOutputString := CONCAT(sOutputString, FB_EXTRACT_HEX_AND_FLIP(PacketAddress + nCounter, 4));
			END_FOR
			
			sOutputString := CONCAT(sOutputString, '$0D$0A');
			
			MEMCPY(ADR(nLastSentPacketID),													// Record the last sent packet ID.
				PacketAddress,
				4);
				
			bLastPacketConfirmed := FALSE;																			// Actually packet prepared.
			eState := E_Communication_Send_States.E_COM_SEND_START_SEND;
			
		E_Communication_Send_States.E_COM_SEND_START_SEND:
			fbSend(	
			cbLen		:= LEN(sOutputString),				// + 1,(* Send string inclusive string (null) delimiter! *)
			pSrc		:= ADR(sOutputString),							(* Address of the string variable *)
			bExecute	:= TRUE);	
			fbTimerSend(IN:=TRUE,PT:=T#500MS);
			IF NOT (fbSend.bBusy) OR fbTimerSend.Q THEN	
				fbTimerSend(IN:=FALSE);
				fbSend(bExecute	:= FALSE);															// Handle errors too.
				eState := E_Communication_Send_States.E_COM_SEND_WAIT_SENT;
			END_IF
			
		E_Communication_Send_States.E_COM_SEND_WAIT_SENT:
			IF nLastReceivedPacketID = nLastSentPacketID THEN
				eState := E_Communication_Send_States.E_COM_SEND_FINALIZE;
			END_IF
			
		E_Communication_Send_States.E_COM_SEND_FINALIZE:	
			bLastPacketConfirmed := TRUE;
																				// Actually packet prepared
	END_CASE
END_IF

END_FUNCTION_BLOCK

// ---- POUs/Mitsubishi/Func/FB_EXTRACT_HEX_AND_FLIP.TcPOU
FUNCTION FB_EXTRACT_HEX_AND_FLIP
VAR_INPUT
	pBytes					: PVOID;																// The address of the bytes array.
	nLenght					: UDINT;																// Number of bytes to be flipped.
END_VAR
VAR_OUTPUT
	sHex					: STRING;																// The value of the extracted and flipped bytes as HEX.
END_VAR
VAR
	sTmpVal					: STRING;																// Medium value.
	nCounter				: UDINT;
END_VAR

sTmpVal := DATA_TO_HEXSTR(pData := pBytes,
cbData := nLenght,
bLoCase := FALSE);
FOR nCounter := 1 TO nLenght BY 1 DO
	sHex := CONCAT(LEFT(sTmpVal, 2), sHex);
	sTmpVal := RIGHT(sTmpVal, LEN(sTmpVal) - 3);
END_FOR

END_FUNCTION

// ---- POUs/Mitsubishi/Sub/FB_SetOutputBuffer.TcPOU
FUNCTION_BLOCK FB_SetOutputBuffer
VAR_INPUT
	OutputBufferAddress				: PVOID;
	PacketAddress					: PVOID;
	SizeOfPacket					: UDINT;
END_VAR
VAR_OUTPUT
	nPacketLenght					: UDINT;
END_VAR
VAR
END_VAR

nPacketLenght := SizeOfPacket;
MEMCPY(OutputBufferAddress, 
		PacketAddress, 
		SizeOfPacket);
		
(*nPacketLenght := nPacketLenght + 1;
MEMSET(OutputBufferAddress + nPacketLenght,
	13,
	1);
	
nPacketLenght := nPacketLenght + 1;
MEMSET(OutputBufferAddress + nPacketLenght,
	10,
	1);
	*)

END_FUNCTION_BLOCK

// ---- POUs/Mitsubishi/Sub/FB_ClearOutputBuffer.TcPOU
FUNCTION_BLOCK FB_ClearOutputBuffer
VAR_INPUT
	OutputBufferAddress				: PVOID;
	SizeOfOutputBuffer				: UDINT;
END_VAR
VAR_OUTPUT
END_VAR
VAR
	NullItem						: BYTE 		:= 0;
END_VAR


MEMSET(OutputBufferAddress,
		NullItem,
		SizeOfOutputBuffer);

END_FUNCTION_BLOCK
